// TIA Portal project "Project1" (V16)

(* hardware
DEVICE "S71500/ET200MP station_1"  S7-1500 station
   slot 0: "Rail_0"  Rack  6ES7 590-1***0-0AA0
   slot 1: "PLC_1"  CPU 1511C-1 PN  6ES7 511-1CK00-0AB0  V2.8
      slot 3: "CPU display_1"  6ES7591-1AA00-0AA0
      slot 32768: "PROFINET interface_1"  X1
         slot 32769: "Port_1"  X1 P1
         slot 32770: "Port_2"  X1 P2
      slot 34817: "Virtual CP interface port_1"  Virtual CP interface port  Virtual CP interface port
*)

// ===== PLC "PLC_1"  CPU 1511C-1 PN =====

VAR_GLOBAL   // PLC tag table "Default tag table"
   "start" AT %I0.0 : Bool;
   "stop" AT %I0.1 : Bool;
   "aa" AT %I0.2 : Bool;
   "sagmotor" AT %Q0.0 : Bool;
   "solmotor" AT %Q0.1 : Bool;
   "yr1" AT %M0.0 : Bool;
END_VAR

// folder: System blocks/Program resources

DATA_BLOCK "bekle1"   // DB5
{ S7_Optimized_Access := 'TRUE' }
AUTHOR : Simatic
FAMILY : IEC
NAME : IEC_TMR
VERSION : 1.0
// stored: InstanceOfName IEC_TIMER
"IEC_TIMER"
BEGIN
END_DATA_BLOCK

DATA_BLOCK "bekle2"   // DB6
{ S7_Optimized_Access := 'TRUE' }
AUTHOR : Simatic
FAMILY : IEC
NAME : IEC_TMR
VERSION : 1.0
// stored: InstanceOfName IEC_TIMER
"IEC_TIMER"
BEGIN
END_DATA_BLOCK

DATA_BLOCK "bekle3"   // DB7
{ S7_Optimized_Access := 'TRUE' }
AUTHOR : Simatic
FAMILY : IEC
NAME : IEC_TMR
VERSION : 1.0
// stored: InstanceOfName IEC_TIMER
"IEC_TIMER"
BEGIN
END_DATA_BLOCK

DATA_BLOCK "bekle4"   // DB8
{ S7_Optimized_Access := 'TRUE' }
AUTHOR : Simatic
FAMILY : IEC
NAME : IEC_TMR
VERSION : 1.0
// stored: InstanceOfName IEC_TIMER
"IEC_TIMER"
BEGIN
END_DATA_BLOCK

// folder: (top level)

ORGANIZATION_BLOCK "Main"   // OB1, LAD, ProgramCycle
TITLE = "Main Program Sweep (Cycle)"
{ S7_Optimized_Access := 'TRUE' }
VERSION : 0.1
   VAR_INPUT
      Initial_Call : Bool;   // Initial call of this OB
      Remanence : Bool;   // =True, if remanent data are available
   END_VAR
   VAR_TEMP   // added for the SCL form of the ladder/FBD networks
      _w1 : Bool;
   END_VAR
BEGIN

REGION Network 1
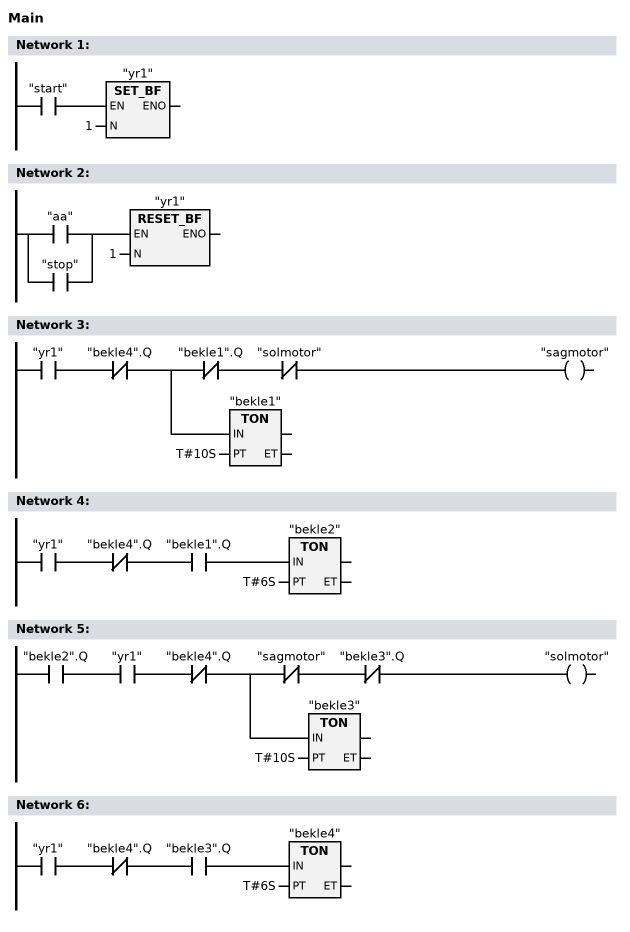
   // no SCL statement known for SBitfield: written as a call
   IF "start" THEN SET_BF(operand := "yr1", n := 1); END_IF;
END_REGION

REGION Network 2
   // no SCL statement known for RBitfield: written as a call
   IF "aa" OR "stop" THEN RESET_BF(operand := "yr1", n := 1); END_IF;
END_REGION

REGION Network 3
   #_w1 := "yr1" AND NOT "bekle4".Q;
   "sagmotor" := #_w1 AND NOT "bekle1".Q AND NOT "solmotor";
   "bekle1".TON(IN := #_w1, PT := T#10S);
END_REGION

REGION Network 4
   "bekle2".TON(IN := "yr1" AND NOT "bekle4".Q AND "bekle1".Q, PT := T#6S);
END_REGION

REGION Network 5
   #_w1 := "bekle2".Q AND "yr1" AND NOT "bekle4".Q;
   "solmotor" := #_w1 AND NOT "sagmotor" AND NOT "bekle3".Q;
   "bekle3".TON(IN := #_w1, PT := T#10S);
END_REGION

REGION Network 6
   "bekle4".TON(IN := "yr1" AND NOT "bekle4".Q AND "bekle3".Q, PT := T#6S);
END_REGION
END_ORGANIZATION_BLOCK